// TwinCAT 3 PLC project Untitled1
// ProgramVersion: 3.1.4026.11
// CompilerDefines: VISU_USEPROPERTYINFO
// libraries:
//   Tc2_Standard, * (Beckhoff Automation GmbH)
//   Tc2_System, * (Beckhoff Automation GmbH)
//   VisuDialogs, * (System)
// project tree:
//   DUTs/ Conveyor.TcDUT
//   / GlobalTextList.TcGTLO, PlcTask.TcTTO, Visualization Manager.TcVMO (not stored)
//   POUs/ ConvState.TcPOU, Flash.TcPOU, MAIN.TcPOU
//   VISUs/ Visualization.TcVIS
// real-time tasks:
//   TASK PlcTask: cycle T#10ms, priority 20, ADS port 350

CONFIGURATION Untitled1
    RESOURCE PLC ON TwinCAT3
        TASK PlcTask(INTERVAL := T#10ms, PRIORITY := 20);
        PROGRAM MAIN WITH PlcTask : MAIN;
    END_RESOURCE
END_CONFIGURATION

// ---- DUTs/Conveyor.TcDUT
TYPE Conveyor :
STRUCT
	//start : BOOL;
	is_started :  BOOL;
	status : INT;
	id : INT;
    red_light_on : BOOL;
    yellow_light_on : BOOL;
    green_light_on : BOOL;
    in_sensor : BOOL;
    out_sensor : BOOL;
    motor_on : BOOL;
	stop : BOOL;
//	was_stopped : BOOL;
	test_lights : BOOL;
	transfer : BOOL;
END_STRUCT
END_TYPE

// ---- POUs/MAIN.TcPOU
PROGRAM MAIN
VAR
conv1 AT %Q* : Conveyor := (
	is_started:=FALSE,
	status:=0, 
	id:=1, 
	red_light_on:=0, 
	yellow_light_on:=0,
	green_light_on:=0,
	in_sensor := 0,
	out_sensor := 0,
	motor_on := 0,
	transfer := 0
);

conv2 : Conveyor := (
	is_started:=0,
	status:=0, 
	id:=2, 
	red_light_on:=0, 
	yellow_light_on:=0,
	green_light_on := 0,
	in_sensor := 0,
	out_sensor := 0,
	motor_on := 0,
	transfer := 0
);

conv3 : Conveyor := (
	is_started:=0,
	status:=0, 
	id:=3, 
	red_light_on:=0, 
	yellow_light_on:=0,
	green_light_on := 0,
	in_sensor := 0,
	out_sensor := 0,
	motor_on := 0,
	transfer := 0
);

	conv1State: ConvState;
	conv2State: ConvState;
	conv3State: ConvState;
END_VAR

conv1State(conv:=conv1);
conv1 := conv1State.conv;

conv2State(conv:=conv2);
conv2 := conv2State.conv;

conv3State(conv:=conv3);
conv3 := conv3State.conv;

END_PROGRAM

// ---- POUs/ConvState.TcPOU
FUNCTION_BLOCK ConvState
VAR_INPUT
	conv: Conveyor;
END_VAR
VAR_OUTPUT
END_VAR
VAR
	fbFlash: Flash;
	Count : INT :=0;
	prevFlashOut: BOOL;
END_VAR

IF conv.stop THEN
	conv.status := 1;
ELSIF conv.test_lights THEN
	conv.status := 4;
ELSIF conv.is_started THEN
	IF (conv.in_sensor OR conv.motor_on) AND conv.transfer THEN
		conv.status := 3;
	ELSE
		conv.status := 2;
	END_IF
ELSE
	conv.status := 0;
END_IF



CASE conv.status OF
	0: // defined default state
		conv.green_light_on := FALSE;
		conv.yellow_light_on := FALSE;
		conv.red_light_on := FALSE;
		conv.motor_on := FALSE;
		//conv.in_sensor := FALSE;
		//conv.out_sensor := FALSE;
			

	1: //red light - stop
		 fbFlash(bstart:=TRUE, Time_off:=T#2S, Time_on:=T#1S);
		 conv.red_light_on := fbFlash.out;
		 conv.motor_on:=FALSE;
		 conv.green_light_on := FALSE;
		 conv.yellow_light_on := FALSE;
		 conv.transfer := FALSE;

		 
	2: //yellow light - idle
		 conv.yellow_light_on := TRUE;
		 conv.red_light_on := FALSE;
		 conv.green_light_on := FALSE;
		 
	3: //green light - running
		 fbFlash(bstart:=TRUE, Time_off:=T#0.5S, Time_on:=T#1S);
		 conv.green_light_on := fbFlash.out;
		 conv.red_light_on := FALSE;
		 conv.yellow_light_on := FALSE;
		 conv.motor_on:=TRUE;
		 
		 IF conv.out_sensor THEN
			 conv.motor_on:=FALSE;
			 conv.transfer:=FALSE;
		 END_IF
		
	4: //test lights
		 fbFlash(bstart:=TRUE, Time_off:=T#0.5S, Time_on:=T#1S);
		 conv.green_light_on := fbFlash.out;
		 conv.red_light_on := fbFlash.out;
		 conv.yellow_light_on := fbFlash.out;
		 conv.motor_on:=FALSE;
		 
		 IF fbFlash.out AND NOT prevFlashOut THEN
    		Count := Count + 1;  // Increment the counter
		 END_IF
		 
		 prevFlashOut := fbFlash.out;
		 
		 IF Count > 5 THEN
			 conv.status := 0;
			 conv.test_lights:= FALSE;
			 Count := 0;
		 END_IF

END_CASE

END_FUNCTION_BLOCK

// ---- POUs/Flash.TcPOU
FUNCTION_BLOCK Flash
VAR
	ton1: TON;
	ton2: TON;
END_VAR
VAR_INPUT
	bstart: BOOL;
	Time_off: TIME;
	Time_on: TIME;
END_VAR
VAR_OUTPUT
	out: BOOL;
END_VAR

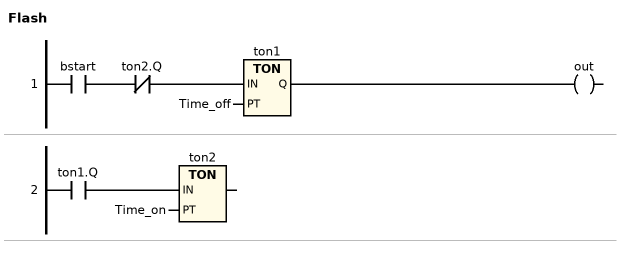
// NETWORK 1
ton1(IN := bstart AND NOT ton2.Q, PT := Time_off); // TON
out := ton1.Q;

// NETWORK 2
ton2(IN := ton1.Q, PT := Time_on); // TON

END_FUNCTION_BLOCK

// ---- GlobalTextList.TcGTLO
TEXTLIST GlobalTextList
  589 = 'Conveyor 1'
  916 = 'Conveyor 2'
  105 = 'Conveyor 3'
  574 = 'in_sensor'
  150 = 'out_sensor'
  925 = 'stop'
END_TEXTLIST

// ---- VISUs/Visualization.TcVIS
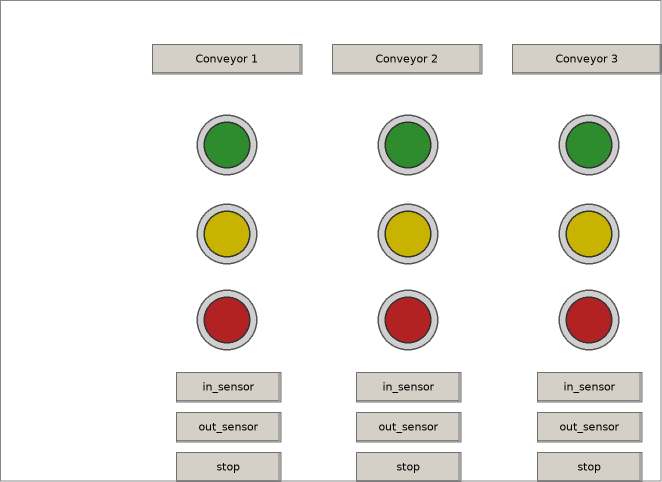
VISUALIZATION Visualization  // 662x482
    Lamp1 (192,285 70x70), variable: MAIN.conv1.red_light_on, style: Lamp-Lamp1-Red
    Lamp1 (192,199 70x70), variable: MAIN.conv1.yellow_light_on, style: Lamp-Lamp1-Yellow
    Lamp1 (192,110 70x70), variable: MAIN.conv1.green_light_on, style: Lamp-Lamp1-Green
    Lamp1 (373,285 70x70), variable: MAIN.conv2.red_light_on, style: Lamp-Lamp1-Red
    Lamp1 (373,199 70x70), variable: MAIN.conv2.yellow_light_on, style: Lamp-Lamp1-Yellow
    Lamp1 (373,110 70x70), variable: MAIN.conv2.green_light_on, style: Lamp-Lamp1-Green
    Lamp1 (554,285 70x70), variable: MAIN.conv3.red_light_on, style: Lamp-Lamp1-Red
    Lamp1 (554,199 70x70), variable: MAIN.conv3.yellow_light_on, style: Lamp-Lamp1-Yellow
    Lamp1 (554,110 70x70), variable: MAIN.conv3.green_light_on, style: Lamp-Lamp1-Green
    Button (176,372 105x30), "in_sensor"
        toggle MAIN.conv1.in_sensor
    Button (176,412 105x30), "out_sensor"
        toggle MAIN.conv1.out_sensor
    Button (356,372 105x30), "in_sensor"
        toggle MAIN.conv2.in_sensor
    Button (356,412 105x30), "out_sensor"
        toggle MAIN.conv2.out_sensor
        OnMouseClick: toggle MAIN.conv2.out_sensor
    Button (537,372 105x30), "in_sensor"
        toggle MAIN.conv3.in_sensor
    Button (537,412 105x30), "out_sensor"
        toggle MAIN.conv3.out_sensor
    Button (176,452 105x30), "stop"
        toggle MAIN.conv1.stop
    Button (356,452 105x30), "stop"
        toggle MAIN.conv2.stop
    Button (537,452 105x30), "stop"
        toggle MAIN.conv3.stop
    Button (152,44 150x30), "Conveyor 1"
        toggle MAIN.conv1.is_started
    Button (332,44 150x30), "Conveyor 2"
        toggle MAIN.conv2.is_started
    Button (512,44 150x30), "Conveyor 3"
        toggle MAIN.conv3.is_started
END_VISUALIZATION
